{attribute 'qualified_only' := ''}
{attribute 'strict' := ''}
TYPE MC_COMBINE_MODE :
(
	enum_member := 0
);
END_TYPE

(* stored: Version 1.1.0.1, ProductVersion 3.1.4024.11
   DUT MC_COMBINE_MODE: Id {5b848e59-e6d7-42ab-a8a4-c6de805ca85e} *)
